                                            ELSIF (instMoveRelative.Error = TRUE) THEN
                                                statResetIncJog := TRUE;
                                                // Errorhandling
                                                statStatus                    := ERR_MC_MOVERELATIVE;
                                                statErrorAutoCleared          := TRUE;
                                                diagnostics                   := statDiagnostics;
                                                diagnostics.subfunctionStatus := instMoveRelative.ErrorId;
                                                // Set next state
                                                statFBState          := AXIS_STOP_ON_ERROR_SELECTION;
                                                statBasicMotionState := NO_SELECTION;
                                                statExeOfBasicMotion := CMD_ERROR;
                                                statIncJogSubState   := INC_JOG_IDLE;

                                            ELSIF (instMoveRelative.CommandAborted = TRUE) THEN
                                                statResetIncJog      := TRUE;
                                                statExeOfBasicMotion := CMD_ABORTED;
                                                statIncJogSubState   := INC_JOG_IDLE;

                                            ELSE
                                                // statJogDistance :=  axis.StatusPositioning.Distance;
                                                ; // Wait for next state
                                            END_IF;

                                        INC_JOG_STOP: // Executed if inputs are reset --> Stop jog operation OR if jogForward and jogBackward are set --> Error and stop axis
                                            instHalt(Axis := axis,
                                                     Execute := TRUE,
                                                     Deceleration := statDeceleration,
                                                     (*AbortAcceleration := FALSE,*)
                                                     Jerk := statJerk);

                                            // Evaluate MC_Command
                                            IF (instHalt.Done = TRUE) THEN
                                                // Set next state
                                                statExeOfBasicMotion := CMD_END_PROCESS;
                                                statIncJogSubState   := INC_JOG_IDLE;

                                            ELSIF (instHalt.Error = TRUE) THEN
                                                statResetIncJog := TRUE;
                                                // Errorhandling
                                                statStatus                    := ERR_MC_HALT;
                                                statErrorAutoCleared          := TRUE;
                                                diagnostics                   := statDiagnostics;
                                                diagnostics.subfunctionStatus := instHalt.ErrorId;
                                                // Set next state
                                                statFBState          := AXIS_STOP_ON_ERROR_SELECTION;
                                                statBasicMotionState := NO_SELECTION;
                                                statExeOfBasicMotion := CMD_ERROR;
                                                statIncJogSubState   := INC_JOG_IDLE;

                                            ELSIF (instHalt.CommandAborted = TRUE) THEN
                                                statResetIncJog := TRUE;
                                                // Set next state
                                                statIncJogSubState   := INC_JOG_IDLE;
                                                statExeOfBasicMotion := CMD_ABORTED;

                                            ELSE
                                                ; // Wait for stopping axis
                                            END_IF;

                                    ELSE
                                        // Errorhandling
                                        statStatus                    := ERR_UNDEFINED_INCREMENTAL_JOG_SUBSTATE;
                                        statErrorUserCleared          := TRUE;
                                        diagnostics                   := statDiagnostics;
                                        diagnostics.subfunctionStatus := 0;
                                        // Set errorstate
                                        statFBState := FB_ERROR;
                                    END_CASE;

                                CMD_DONE,
                                    CMD_ABORTED,
                                    CMD_ERROR,
                                    CMD_END_PROCESS:
                                    // Return to NO_SELECTION if command finished
                                    IF (statBasicCommand.2 = FALSE) AND (statBasicCommand.3 = FALSE)
                                        THEN
                                        // jogForward and jogbackward inputs are reset
                                        statExeOfBasicMotion := CMD_BUSY;
                                        statBasicMotionState := NO_SELECTION;
                                    ELSE
                                        ; // Wait for falling edge at inputs for jog
                                    END_IF;

                            ELSE
                                // Errorhandling
                                statStatus                    := ERR_UNDEFINED_INCREMENTAL_JOG_STATE;
                                statErrorUserCleared          := TRUE;
                                diagnostics.subfunctionStatus := 0;
                                diagnostics.basicMotionState  := statBasicMotionState;
                                // Set errorstate
                                statFBState := FB_ERROR;
                            END_CASE;
                    {END_REGION}

                    ELSE
                        // Errorhandling - Invalid jog state
                        statStatus                    := ERR_INVALID_JOG_MODE;
                        statErrorAutoCleared          := TRUE;
                        diagnostics                   := statDiagnostics;
                        diagnostics.subfunctionStatus := 0;
                        // Set next state
                        statFBState          := AXIS_STOP_ON_ERROR_SELECTION;
                        statBasicMotionState := NO_SELECTION;
                    END_CASE;
                {END_REGION}

                MOVE_VELOCITY_SELECTED:
                    // Additional features (applicative): Change setpoint on the fly (Velocity) 
                    {REGION "MOVEVELOCITY_SELECTED"}

                    // Firstcycle of command
                    IF (statFirstCycleBasicMotion = TRUE) THEN
                        // Reset MC_MOVEVELOCITY command
                        instMoveVelocity(Axis := axis,
                                         Execute := FALSE);

                        statVelocityChangeOnTheFly := configuration.moveVelocity.velocityChangeOnTheFly;
                        statVelocity               := configuration.moveVelocity.velocity;           // Store the last adjusted velocity value
                        statAcceleration           := configuration.moveVelocity.acceleration;       // Store the last adjusted acceleration value
                        statDeceleration           := configuration.moveVelocity.deceleration;       // Store the last adjusted deceleration value
                        statJerk                   := configuration.moveVelocity.jerk;               // Store the last adjusted jerk value 
                        statDirection              := configuration.moveVelocity.direction;          // Store the last adjusted axis direction 
                        statPositionControlled     := configuration.moveVelocity.positionControlled; // Store the last adjusted motion mode

                    ELSIF (statVelocityChangeOnTheFly = TRUE) AND
                        (configuration.moveVelocity.velocity <> statVelocity) // Velocity changed
                        AND
                        (instMoveVelocity.CommandAborted = FALSE)
                        THEN
                        // Reset MC_MOVEVELOCITY command
                        instMoveVelocity(Axis := axis,
                                         Execute := FALSE);

                        statVelocity := configuration.moveVelocity.velocity; // Store the last adjusted velocity value
                    END_IF;

                    // Call MC_Command
                    instMoveVelocity(Axis := axis,
                                     Execute := statBasicCommand.4 OR statFirstCycleBasicMotion, // Input: moveVelocity
                                     Velocity := statVelocity,
                                     Acceleration := statAcceleration,
                                     Deceleration := statDeceleration,
                                     Jerk := statJerk,
                                     Direction := statDirection,
                    (*PositionControlled :=  statPositionControlled,*)
                    (*Current := FALSE*) );

                    // Evaluate MC_Command
                    IF (instMoveVelocity.Busy = FALSE) AND
                        (instMoveVelocity.Error = FALSE) AND
                        (instMoveVelocity.CommandAborted = FALSE) AND
                        (instMoveVelocity.InVelocity = FALSE)
                        THEN
                        // Return to NO_SELECTION if command finished
                        statBasicMotionState := NO_SELECTION;

                    ELSIF (instMoveVelocity.Error = TRUE)
                        THEN
                        // Errorhandling
                        statStatus                    := ERR_MC_MOVEVELOCITY;
                        statErrorAutoCleared          := TRUE;
                        diagnostics                   := statDiagnostics;
                        diagnostics.subfunctionStatus := instMoveVelocity.ErrorId;
                        statVelocityChangeOnTheFly    := FALSE;
                        // Set next state
                        statFBState          := AXIS_STOP_ON_ERROR_SELECTION;
                        statBasicMotionState := NO_SELECTION;

                    ELSE
                        ; // Command selected
                    END_IF;

                    // Write MC_Command outputs to internal variable
                    statExeOfBasicMotion   := 16#0;
                    statExeOfBasicMotion.0 := instMoveVelocity.Busy;
                    statExeOfBasicMotion.2 := instMoveVelocity.CommandAborted;
                    statExeOfBasicMotion.3 := instMoveVelocity.Error;
                    statExeOfBasicMotion.4 := instMoveVelocity.InVelocity;
                {END_REGION}

                POS_RELATIVE_SELECTED:
                    // Additional features (applicative): Specified direction
                    {REGION "POS_RELATIVE_SELECTED"}
                    // Firstcycle of command
                    IF (statFirstCycleBasicMotion = TRUE) THEN
                        // Configurate the direction of rotation
                        // 
                        IF ((configuration.posRelative.direction = 0) AND (configuration.posRelative.distance >= 0.0)
                            ) // Sign of distance is evaluated
                            OR
                            (configuration.posRelative.direction = FORWARD_DIR) // Forward direction
                            THEN
                            statPosition := ABS(configuration.posRelative.distance);
                            // Reset MC_MOVERELATIVE command
                            instMoveRelative(Axis := axis,
                                             Execute := FALSE);

                            statApplicativeBasicMotionError := FALSE;

                        ELSIF ((configuration.posRelative.direction = 0) AND (configuration.posRelative.distance < 0.0)
                            ) // Sign of distance is evaluated
                            OR
                            (configuration.posRelative.direction = BACKWARD_DIR) // Backward direction
                            THEN
                            statPosition := -ABS(configuration.posRelative.distance);
                            // Reset MC_MOVERELATIVE command
                            instMoveRelative(Axis := axis,
                                             Execute := FALSE);

                            statApplicativeBasicMotionError := FALSE;

                        ELSE
                            // Errorhandling - Invalid direction
                            statStatus                      := ERR_INVALID_POS_RELATIVE_DIR;
                            statErrorAutoCleared            := TRUE;
                            diagnostics.subfunctionStatus   := 0;
                            diagnostics                     := statDiagnostics;
                            statApplicativeBasicMotionError := TRUE;
                            // Set next state
                            statFBState          := AXIS_STOP_ON_ERROR_SELECTION;
                            statBasicMotionState := NO_SELECTION;
                        END_IF;
                    END_IF;

                    IF (statApplicativeBasicMotionError = FALSE) THEN
                        // Call MC_Command
                        instMoveRelative(Axis := axis,
                                         Execute := statBasicCommand.5 OR statFirstCycleBasicMotion, // Input: posRelative
                                         Distance := statPosition,
                                         Velocity := configuration.posRelative.velocity,
                                         Acceleration := configuration.posRelative.acceleration,
                                         Deceleration := configuration.posRelative.deceleration,
                                         Jerk := configuration.posRelative.jerk);

                        // Evaluate MC_Command
                        IF (instMoveRelative.Busy = FALSE) AND
                            (instMoveRelative.Error = FALSE) AND
                            (instMoveRelative.Done = FALSE) AND
                            (instMoveRelative.CommandAborted = FALSE)
                            THEN
                            // Return to NO_SELECTION if command finished
                            statBasicMotionState := NO_SELECTION;

                        ELSIF (instMoveRelative.Error = TRUE) THEN
                            // Errorhandling
                            statStatus                    := ERR_MC_MOVERELATIVE;
                            statErrorAutoCleared          := TRUE;
                            diagnostics                   := statDiagnostics;
                            diagnostics.subfunctionStatus := instMoveRelative.ErrorId;
                            // Set next state
                            statFBState          := AXIS_STOP_ON_ERROR_SELECTION;
                            statBasicMotionState := NO_SELECTION;
                        ELSE
                            ; // Command selected
                        END_IF;

                        // Write MC_Command outputs to internal variable
                        statExeOfBasicMotion   := 16#0;
                        statExeOfBasicMotion.0 := instMoveRelative.Busy;
                        statExeOfBasicMotion.1 := instMoveRelative.Done;
                        statExeOfBasicMotion.2 := instMoveRelative.CommandAborted;
                        statExeOfBasicMotion.3 := instMoveRelative.Error;

                    ELSE
                        ; // Direction not valid
                    END_IF;
                {END_REGION}

                POS_ABSOLUTE_SELECTED:
                    // Additional features (applicative): Change setpoint on the fly (Velocity and Position)
                    {REGION "POS_ABSOLUTE_SELECTED"}
                    // Firstcycle of command
                    IF (statFirstCycleBasicMotion = TRUE) THEN
                        // Reset MC_MOVEABSOLUTE command
                        instMoveAbsolute(Axis := axis,
                                         Execute := FALSE);

                        statPosition     := configuration.posAbsolute.position;
                        statVelocity     := configuration.posAbsolute.velocity;     // Store the last adjusted velocity value
                        statAcceleration := configuration.posAbsolute.acceleration; // Store the last adjusted accerlation value
                        statDeceleration := configuration.posAbsolute.deceleration; // Store the last adjusted deceleration value
                        statJerk         := configuration.posAbsolute.jerk;         // Store the last adjusted jerk value
                        statDirection    := configuration.posAbsolute.direction;

                        statVelocityChangeOnTheFly := configuration.posAbsolute.velocityChangeOnTheFly;
                        statPositionChangeOnTheFly := configuration.posAbsolute.positionChangeOnTheFly;

                    ELSIF (((statVelocityChangeOnTheFly = TRUE) AND (configuration.posAbsolute.velocity <> statVelocity)) OR
                        ((statPositionChangeOnTheFly = TRUE) AND (configuration.posAbsolute.position <> statPosition))) AND
                        (instMoveAbsolute.CommandAborted = FALSE)
                        THEN
                        instMoveAbsolute(Axis := axis,
                                         Execute := FALSE);

                        IF (statVelocityChangeOnTheFly = TRUE) THEN // Apply the new velocity value
                            statVelocity := configuration.posAbsolute.velocity;
                        END_IF;

                        IF (statPositionChangeOnTheFly = TRUE) THEN // Apply the new position value
                            statPosition := configuration.posAbsolute.position;
                        END_IF;

                        // Reset MC_MOVEABSOLUTE command
                        instMoveAbsolute(Axis := axis,
                                         Execute := FALSE);
                    END_IF;

                    instMoveAbsolute(Axis := axis,
                                     Execute := statBasicCommand.6 OR statFirstCycleBasicMotion, // Input: posAbsolute
                                     Position := statPosition,
                                     Velocity := statVelocity,
                                     Acceleration := statAcceleration,
                                     Deceleration := statDeceleration,
                                     Jerk := statJerk,
                    (*Direction :=  statDirection*) );

                    // Evaluate MC_Command
                    IF (instMoveAbsolute.Busy = FALSE) AND
                        (instMoveAbsolute.Error = FALSE) AND
                        (instMoveAbsolute.Done = FALSE) AND
                        (instMoveAbsolute.CommandAborted = FALSE)
                        THEN
                        // Return to NO_SELECTION if command finished
                        statBasicMotionState := NO_SELECTION;

                    ELSIF (instMoveAbsolute.Error = TRUE) THEN
                        // Errorhandling
                        statStatus                    := ERR_MC_MOVEABSOLUTE;
                        statErrorAutoCleared          := TRUE;
                        diagnostics                   := statDiagnostics;
                        diagnostics.subfunctionStatus := instMoveAbsolute.ErrorId;
                        statVelocityChangeOnTheFly    := FALSE;
                        statPositionChangeOnTheFly    := FALSE;
                        // Set next state
                        statFBState          := AXIS_STOP_ON_ERROR_SELECTION;
                        statBasicMotionState := NO_SELECTION;

                    ELSE
                        ; // Command selected
                    END_IF;

                    // Write MC_Command outputs to internal variable
                    statExeOfBasicMotion   := 16#0;
                    statExeOfBasicMotion.0 := instMoveAbsolute.Busy;
                    statExeOfBasicMotion.1 := instMoveAbsolute.Done;
                    statExeOfBasicMotion.2 := instMoveAbsolute.CommandAborted;
                    statExeOfBasicMotion.3 := instMoveAbsolute.Error;
                {END_REGION}

                ACTIVE_HOMING_SELECTED:
                    // Additional fearure (applicative): homing on fixed stop
                    {REGION "ACTIVE_HOMING_SELECTED"}
                    // Firstcycle of command
                    IF (statFirstCycleBasicMotion = TRUE) THEN
                        statActiveHomingState  := configuration.homing.extendedMode;
                        statExeOfBasicMotion   := CMD_BUSY;
                        statPassiveHomingState := NO_HOMING_ACTIVE;
                    END_IF;

                    // Selection of extended homing mode  
                    CASE statActiveHomingState OF
                        STANDARD_HOMING:
                            // No additional features
                            {REGION "STANDARD_HOMING"}
                            // Firstcycle of command
                            IF (statFirstCycleBasicMotion = TRUE) THEN
                                // Reset MC_HOME command
                                instHome(Axis := axis,
                                         bCalibrationCam := homingSensor,
                                         Execute := FALSE);

                                // Reset TON command
                                instTimerTON(IN := FALSE,
                                             PT := configuration.homing.homeExecutionTimeLimit);
                            END_IF;

                            // Call MC_Command
                            instHome(Axis := axis,
                                     bCalibrationCam := homingSensor,
                                     Execute := statBasicCommand.10 OR statFirstCycleBasicMotion, // Input: homing
                                     Position := configuration.homing.position,
                            (*Mode :=  configuration.homing.mode*) );

                            //Call TON
                            instTimerTON(IN := TRUE,
                                         PT := configuration.homing.homeExecutionTimeLimit);

                            // Evaluate MC_Command
                            IF (instHome.Busy = FALSE) AND
                                (instHome.Done = FALSE) AND
                                (instHome.CommandAborted = FALSE) AND
                                (instHome.Error = FALSE)
                                THEN
                                // Return to NO_SELECTION if command finished
                                statActiveHomingState := STANDARD_HOMING;
                                statBasicMotionState  := NO_SELECTION;

                            ELSIF (instHome.Error = TRUE OR instTimerTON.Q) THEN
                                // Errorhandling
                                statStatus                    := ERR_MC_HOME;
                                statErrorAutoCleared          := TRUE;
                                diagnostics                   := statDiagnostics;
                                diagnostics.subfunctionStatus := instHome.ErrorId;
                                statFBState                   := AXIS_STOP_ON_ERROR_SELECTION;
                                statBasicMotionState          := NO_SELECTION;

                            ELSE
                                ; // Command selected

                            END_IF;

                            statExeOfBasicMotion   := 16#0;
                            statExeOfBasicMotion.0 := instHome.Busy;
                            statExeOfBasicMotion.1 := instHome.Done;
                            statExeOfBasicMotion.2 := instHome.CommandAborted;
                            statExeOfBasicMotion.3 := instHome.Error;
                        {END_REGION}
                        HOMING_ON_FIXED_STOP:
                            // This case is additional feature (MC_MOVEVELOCITY and MC_HOME internal used)
                            {REGION "REFERENCE_TO_FIXED_STOP"}
                            CASE statExeOfBasicMotion OF
                                CMD_BUSY:
                                    // Firstcycle of command
                                    IF (statFirstCycleBasicMotion = TRUE) THEN
                                        // Check if homing on fixed stop is allowed  
                                        (*IF ( axis.Modulo.Enable = TRUE) THEN*)
                                        IF (tempFalse = TRUE) THEN
                                            // Modulo enabled - Errorhandling
                                            statStatus                    := ERR_MODULO_NOT_ALLOWED;
                                            statErrorAutoCleared          := TRUE;
                                            diagnostics.subfunctionStatus := 0;
                                            diagnostics.basicMotionState  := statBasicMotionState;
                                            // Set next state
                                            statFBState           := AXIS_STOP_ON_ERROR_SELECTION;
                                            statBasicMotionState  := NO_SELECTION;
                                            statActiveHomingState := STANDARD_HOMING;
                                            statHomingSubState    := HOMING_IDLE;

                                        ELSIF (configuration.homing.extendedModeTorqueLimit = 0) // Torqueliming 0 in configuration 
                                            THEN
                                            // Errorhandling -  Torquevalue 0 configured
                                            statStatus                    := ERR_INVALID_TORQUE_LIMIT;
                                            statErrorAutoCleared          := TRUE;
                                            diagnostics.subfunctionStatus := 0;
                                            diagnostics.basicMotionState  := statBasicMotionState;
                                            // Set next state
                                            statFBState           := AXIS_STOP_ON_ERROR_SELECTION;
                                            statBasicMotionState  := NO_SELECTION;
                                            statActiveHomingState := STANDARD_HOMING;
                                            statHomingSubState    := HOMING_IDLE;

                                            (*ELSIF ( axis.Homing.ReferencingVelocity = 0)*)
                                        ELSIF (configuration.homing.offsetPositionVelocity = 0)
                                            THEN
                                            // Errorhandling -  Velocity 0 configured
                                            statStatus                    := ERR_INVALID_VELOCITY;
                                            statErrorAutoCleared          := TRUE;
                                            diagnostics.subfunctionStatus := 0;
                                            diagnostics.basicMotionState  := statBasicMotionState;
                                            // Set next state
                                            statFBState           := AXIS_STOP_ON_ERROR_SELECTION;
                                            statBasicMotionState  := NO_SELECTION;
                                            statActiveHomingState := STANDARD_HOMING;
                                            statHomingSubState    := HOMING_IDLE;

                                        ELSE
                                            // Store dynamic values
                                            (*statHomingPosition :=  configuration.homing.position;
	                             statVelocity :=  axis.Homing.ReferencingVelocity;
	                             statAcceleration :=  axis.DynamicDefaults.Acceleration;
	                             statDeceleration :=  axis.DynamicDefaults.Deceleration;
	                             statJerk :=  axis.DynamicDefaults.Jerk;
	                             statTorqueLimit :=  configuration.homing.extendedModeTorqueLimit;*)
                                            statHomingPosition := configuration.homing.position;
                                            statVelocity       := configuration.homing.offsetPositionVelocity;
                                            statAcceleration   := configuration.homing.offsetPositionAcceleration;
                                            statDeceleration   := configuration.homing.offsetPositonDeceleration;
                                            statJerk           := configuration.homing.offsetPositionJerk;
                                            statTorqueLimit    := configuration.homing.extendedModeTorqueLimit;

                                            // Detecting operating sensor
                                            (*
								FOR  tempIndex := 1 TO 4 DO
	                              IF  axis.StatusSensor[ tempIndex].Control = TRUE
	                              THEN
	                                EXIT;
	                              END_IF;
	                            END_FOR;
	                            *)
                                            (*IF ( axis.Sensor[ tempIndex].ActiveHoming.Direction = 0) // Positve direction configured
	                            THEN*)
                                            // Positive direction
                                            statDirection := FORWARD_DIR;
                                            (* ELSE
	                              // Negative direction
	                               statDirection :=  BACKWARD_DIR;
	                            END_IF;
	                            *)
                                            (*statTorqueLimitingState :=  FIXED_STOP_DETECTION_ACTIVE;*)
                                            // Reset MC_Commands
                                            instHome(Axis := axis,
                                                     bCalibrationCam := homingSensor,
                                                     Execute := FALSE);

                                            instMoveVelocity(Axis := axis,
                                                             Execute := FALSE);

                                            instMoveAbsolute(Axis := axis,
                                                             Execute := FALSE);

                                            // Reset TON
                                            instTimerTON(IN := FALSE,
                                                         PT := configuration.homing.homeExecutionTimeLimit);

                                            // Determine the encoder type
                                            (* tempIndex := 1;
	                             tempIndex := UDINT_TO_INT( axis.OperativeSensor);
	                            IF ( axis.Sensor[ tempIndex].Type =  INCREMENTAL_ENCODER) THEN
	                               statHomingMode :=  DIRECT_HOMING; // Direct homing (absolute)
	                            ELSE
	                               statHomingMode :=  ABSOLUTE_ENCODER_ADJUSTMENT;
	                            END_IF;
								*)
                                            // Use always direct homing
                                            // statHomingMode :=  DIRECT_HOMING; // Direct homing (absolute)
                                            // Set next state
                                            (*statHomingSubState :=  HOMING_FIXED_STOP_DETECTION;*)
                                            statHomingSubState := HOMING_PROCESS;
                                        END_IF;
                                    END_IF;

                                    // Call OF subStateMachine
                                    REPEAT
                                        CASE statHomingSubState OF
                                            HOMING_IDLE:
                                                tempStateChangeActive := FALSE;
                                                ; // Do nothing, inserted no exectution of homing if error occurred in first cycle

                                            HOMING_FIXED_STOP_DETECTION:
                                                tempStateChangeActive := FALSE;

                                                // Start axis to detect fixed stop
                                                instMoveVelocity(Axis := axis,
                                                                 Execute := TRUE,
                                                                 Velocity := statVelocity,
                                                                 Acceleration := statAcceleration,
                                                                 Deceleration := statDeceleration,
                                                                 Jerk := statJerk,
                                                (*PositionControlled := TRUE,*)
                                                (*Direction :=  statDirection*) );

                                                // Read Statusword only when not already read out
                                                IF (tempStatusWord = 16#0)
                                                    THEN
                                                    (*tempStatusWord :=  axis.StatusWord;*)
                                                    tempStatusWord := axis.NcToPlc.StateDWord;
                                                END_IF;

                                                // Evaluate MC_Command
                                                IF (tempStatusWord.30 = TRUE) THEN // inClamping = TRUE
                                                    // Fixed stop detected --> start homing process
                                                    statHomingSubState    := HOMING_PROCESS;
                                                    tempStateChangeActive := TRUE;

                                                ELSIF (instMoveVelocity.Error = TRUE) THEN
                                                    // Errorhandling
                                                    statStatus                    := ERR_MC_MOVEVELOCITY;
                                                    statErrorAutoCleared          := TRUE;
                                                    diagnostics                   := statDiagnostics;
                                                    diagnostics.subfunctionStatus := instMoveVelocity.ErrorId;
                                                    // Set next state
                                                    statFBState           := AXIS_STOP_ON_ERROR_SELECTION;
                                                    statBasicMotionState  := NO_SELECTION;
                                                    statActiveHomingState := STANDARD_HOMING;
                                                    statExeOfBasicMotion  := CMD_ERROR;
                                                    statHomingSubState    := HOMING_IDLE;

                                                ELSIF (instMoveVelocity.CommandAborted = TRUE) THEN
                                                    // Set next state
                                                    statExeOfBasicMotion := CMD_ABORTED;
                                                    statHomingSubState   := HOMING_IDLE;

                                                ELSE
                                                    ; // Wait for detecting fixed stop
                                                END_IF;

                                            HOMING_PROCESS:
                                                tempStateChangeActive := FALSE;
                                                // Execute MC_HOME
                                                instHome(Axis := axis,
                                                         bCalibrationCam := homingSensor,
                                                         Execute := TRUE,
                                                         Position := statHomingPosition,
                                                (*Mode :=  statHomingMode*) );

                                                //Call TON
                                                instTimerTON(IN := TRUE,
                                                             PT := configuration.homing.homeExecutionTimeLimit);

                                                // Evaluate MC_Command
                                                IF (instHome.Done = TRUE) THEN
                                                    // MC_HOME finished - Set next state
                                                    statHomingSubState    := HOMING_POSITION;
                                                    tempStateChangeActive := TRUE;
                                                    instTimerTON.IN       := FALSE;

                                                ELSIF (instHome.Error = TRUE OR instTimerTON.Q) THEN
                                                    // Errorhandling
                                                    statStatus                    := ERR_MC_HOME;
                                                    statErrorAutoCleared          := TRUE;
                                                    diagnostics                   := statDiagnostics;
                                                    diagnostics.subfunctionStatus := instHome.ErrorId;
                                                    // Set next state
                                                    statFBState          := AXIS_STOP_ON_ERROR_SELECTION;
                                                    statExeOfBasicMotion := CMD_ERROR;
                                                    statHomingSubState   := HOMING_IDLE;

                                                ELSIF (instHome.CommandAborted = TRUE) THEN
                                                    // Set next state
                                                    statExeOfBasicMotion := CMD_ABORTED;
                                                    statHomingSubState   := HOMING_IDLE;
                                                ELSE
                                                    ; // Wait for finish homing process
                                                END_IF;

                                            HOMING_POSITION:
                                                tempStateChangeActive := FALSE;

                                                statHomingPosition := configuration.homing.offsetPosition;
                                                statVelocity       := configuration.homing.offsetPositionVelocity;
                                                statAcceleration   := configuration.homing.offsetPositionAcceleration;
                                                statDeceleration   := configuration.homing.offsetPositonDeceleration;
                                                statJerk           := configuration.homing.offsetPositionJerk;

                                                // Execute moving to homeposition
                                                instMoveAbsolute(Axis := axis,
                                                                 Execute := TRUE,
                                                                 (*Position :=  statHomingPosition,*)
                                                                 Position := configuration.homing.offsetPosition,
                                                                 Velocity := ABS(statVelocity),
                                                                 Acceleration := statAcceleration,
                                                                 Deceleration := statDeceleration,
                                                                 Jerk := statJerk,
                                                (*Direction :=  SHORTEST_WAY_DIR*) );

                                                // Evaluate MC_Command
                                                IF (instMoveAbsolute.Done = TRUE) THEN
                                                    // Homeposition reached - Set next state
                                                    statExeOfBasicMotion := CMD_DONE;
                                                    statHomingSubState   := HOMING_IDLE;

                                                ELSIF (instMoveAbsolute.Error = TRUE) THEN
                                                    // Errorhandling
                                                    statStatus                    := ERR_MC_MOVEABSOLUTE;
                                                    statErrorAutoCleared          := TRUE;
                                                    diagnostics                   := statDiagnostics;
                                                    diagnostics.subfunctionStatus := instMoveAbsolute.ErrorId;
                                                    // Set next state
                                                    statFBState           := AXIS_STOP_ON_ERROR_SELECTION;
                                                    statBasicMotionState  := CMD_BUSY;
                                                    statActiveHomingState := STANDARD_HOMING;
                                                    statExeOfBasicMotion  := CMD_ERROR;
                                                    statHomingSubState    := HOMING_IDLE;

                                                ELSIF (instMoveAbsolute.CommandAborted = TRUE) THEN
                                                    // Set next state
                                                    statExeOfBasicMotion := CMD_ABORTED;
                                                    statHomingSubState   := HOMING_IDLE;

                                                ELSE
                                                    ; // Wait for reaching homeposition
                                                END_IF;

                                        ELSE
                                            // Errorhandling 
                                            statStatus                    := ERR_UNDEFINED_EXTENDED_HOMING_SUBSTATE;
                                            statErrorUserCleared          := TRUE;
                                            diagnostics                   := statDiagnostics;
                                            diagnostics.subfunctionStatus := 0;
                                            // Set errorstate
                                            statFBState           := FB_ERROR;
                                            tempStateChangeActive := FALSE;
                                        END_CASE;

                                    UNTIL (tempStateChangeActive = FALSE) // Repeat execution if a state is changing
                                    END_REPEAT;

                                CMD_DONE,
                                    CMD_ABORTED,
                                    CMD_ERROR:
                                    // Return to NO_SELECTION if command finished
                                    IF (statBasicCommand.10 = FALSE) // homing = FALSE
                                        THEN
                                        // Return to NO_HOMING_ACTIVE if command finished
                                        statBasicMotionState  := NO_SELECTION;
                                        statActiveHomingState := STANDARD_HOMING;
                                        statExeOfBasicMotion  := CMD_BUSY;
                                        statHomingSubState    := HOMING_IDLE;
                                    ELSE
                                        ; // Wait for falling edge at homing command
                                    END_IF;

                            ELSE
                                // Errorhandling
                                statStatus                    := ERR_UNDEFINED_EXTENDED_HOMING_STATE;
                                statErrorUserCleared          := TRUE;
                                diagnostics                   := statDiagnostics;
                                diagnostics.subfunctionStatus := 0;
                                // Set errorstate
                                statFBState := FB_ERROR;
                            END_CASE;
                    {END_REGION}

                    ELSE
                        // Errorhandling
                        statStatus                    := ERR_INVALID_HOMING_EXTENDED_MODE;
                        statErrorAutoCleared          := TRUE;
                        diagnostics                   := statDiagnostics;
                        diagnostics.subfunctionStatus := 0;
                        // Set next state
                        statFBState           := AXIS_STOP_ON_ERROR_SELECTION;
                        statBasicMotionState  := NO_SELECTION;
                        statActiveHomingState := STANDARD_HOMING;
                        statBasicMotionState  := NO_SELECTION;
                    END_CASE;
                {END_REGION}

                GEAR_IN_RELATIVE_SELECTED:
                    // Additional features (applicative): Change setpoint on the fly (gear ratio)
                    {REGION "GEAR_IN_RELATIVE_SELECTED"}
                    // Firstcycle of command
                    IF (statFirstCycleBasicMotion = TRUE) THEN
                        // Reset GEAR_IN command 
                        instGearIn(Master := master,
                                   Slave := axis,
                                   Execute := FALSE);

                        (*statRatioNumerator :=  configuration.gearInRelative.ratioNumerator;*)
                        statRatioNumerator      := configuration.gearInRelative.ratioDenominator;
                        statRatioDenominator    := configuration.gearInRelative.ratioDenominator;
                        statAcceleration        := configuration.gearInRelative.acceleration;
                        statDeceleration        := configuration.gearInRelative.deceleration;
                        statJerk                := configuration.gearInRelative.jerk;
                        statRatioChangeOnTheFly := configuration.gearInRelative.ratioChangeOnTheFly;

                    ELSIF ((statRatioChangeOnTheFly = TRUE) // Flying change of ratio numerator
                    (*AND (( configuration.gearInRelative.ratioNumerator <>  statRatioNumerator)*)
                        AND
                        ((configuration.gearInRelative.ratioDenominator <> statRatioNumerator) OR
                        (configuration.gearInRelative.ratioDenominator <> statRatioDenominator))) AND
                        (instGearIn.CommandAborted = FALSE)
                        THEN
                        instGearIn(Master := master,
                                   Slave := axis,
                                   Execute := FALSE);

                        statRatioNumerator   := configuration.gearInRelative.ratioDenominator; // Apply the new gear ratio numerator
                        statRatioDenominator := configuration.gearInRelative.ratioDenominator; // Apply the new gear ratio denominator
                    END_IF;

                    // Call MC_Command
                    instGearIn(Master := master,
                               Slave := axis,
                               Execute := statBasicCommand.7 OR statFirstCycleBasicMotion, // Input: gearInRelative
                               RatioNumerator := statRatioNumerator,
                               RatioDenominator := DINT_TO_UINT(statRatioDenominator),
                               Acceleration := statAcceleration,
                               Deceleration := statDeceleration,
                               Jerk := statJerk);

                    // Evaluate MC_Command
                    IF (instGearIn.Busy = FALSE) AND
                        (instGearIn.Error = FALSE) AND
                        (instGearIn.CommandAborted = FALSE) AND
                        (instGearIn.InGear = FALSE)
                        THEN
                        // Return to NO_SELECTION if command finished
                        statBasicMotionState := NO_SELECTION;

                    ELSIF (instGearIn.Error = TRUE) THEN
                        // Errorhandling
                        statStatus                    := ERR_MC_GEARIN;
                        statErrorAutoCleared          := TRUE;
                        diagnostics                   := statDiagnostics;
                        diagnostics.subfunctionStatus := instGearIn.ErrorId;
                        statRatioChangeOnTheFly       := FALSE;
                        // Set next state
                        statFBState          := AXIS_STOP_ON_ERROR_SELECTION;
                        statBasicMotionState := NO_SELECTION;

                    ELSE
                        ; // Command selected
                    END_IF;

                    // Read Statusword only when not already read out
                    // IF ( tempStatusWord = 16#0)
                    // THEN
                    //    tempStatusWord :=  axis.StatusWord;
                    // END_IF;

                    // Write MC_Command outputs to internal variable
                    statExeOfBasicMotion   := 16#0;
                    statExeOfBasicMotion.0 := instGearIn.Busy;
                    statExeOfBasicMotion.2 := instGearIn.CommandAborted;
                    statExeOfBasicMotion.3 := instGearIn.Error;
                    // statExeOfBasicMotion.6 :=  tempStatusWord.21 AND NOT  instGearIn.InGear; // write Synchronizing only when bit of instance of MC_GearIn.InGear = FALSE
                    statExeOfBasicMotion.7 := instGearIn.InGear;
                {END_REGION}

                GEAR_IN_ABSOLUTE_SELECTED:
                    // Additional features (applicative): Change setpoint on the fly (gear ratio)
                    {REGION "GEAR_IN_SELECTED"}
                    // Firstcycle of command
                    IF (statFirstCycleBasicMotion = TRUE) THEN
                        // Reset GEAR_IN_POS command 
                        instGearInPos(Master := master,
                                      Slave := axis,
                        (*Execute := FALSE*) );

                        statRatioNumerator       := configuration.gearInAbsolute.ratioNumerator;
                        statRatioDenominator     := configuration.gearInAbsolute.ratioDenominator;
                        statMasterSyncPosition   := configuration.gearInAbsolute.masterSyncPosition;
                        statSlaveSyncPosition    := configuration.gearInAbsolute.slaveSyncPosition;
                        statSyncProfileReference := configuration.gearInAbsolute.syncProfileReference;
                        statMasterStartDistance  := configuration.gearInAbsolute.masterStartDistance;
                        statVelocity             := configuration.gearInAbsolute.velocity;
                        statAcceleration         := configuration.gearInAbsolute.acceleration;
                        statDeceleration         := configuration.gearInAbsolute.deceleration;
                        statJerk                 := configuration.gearInAbsolute.jerk;
                        statSyncDirection        := configuration.gearInAbsolute.syncDirection;
                        statRatioChangeOnTheFly  := configuration.gearInAbsolute.ratioChangeOnTheFly;

                    ELSIF (((statRatioChangeOnTheFly = TRUE) AND (configuration.gearInAbsolute.ratioNumerator <> statRatioNumerator)) OR
                        ((statRatioChangeOnTheFly = TRUE) AND (configuration.gearInAbsolute.ratioDenominator <> statRatioDenominator))) AND
                        (instGearInPos.CommandAborted = FALSE)
                        THEN
                        instGearInPos(Master := master,
                                      Slave := axis,
                        (*Execute := FALSE*) );

                        statRatioNumerator   := configuration.gearInAbsolute.ratioNumerator;   // Apply the new gear ratio numerator
                        statRatioDenominator := configuration.gearInAbsolute.ratioDenominator; // Apply the new gear ratio denominator
                    END_IF;

                    // Call MC_Command
                    instGearInPos(Master := master,
                                  Slave := axis,
                                  Enable := statBasicCommand.8 OR statFirstCycleBasicMotion, // Input: gearInAbsolute
                                  GearRatio := statRatioNumerator,
                                  (*RatioDenominator :=  statRatioDenominator,*)
                                  (*MasterSyncPosition :=  statMasterSyncPosition,*)
                                  (*SlaveSyncPosition :=  statSlaveSyncPosition,*)
                                  (*SyncProfileReference :=  statSyncProfileReference,*)
                                  (*MasterStartDistance :=  statMasterStartDistance,*)
                                  (*Velocity :=  statVelocity,*)
                                  (*Acceleration :=  statAcceleration,*)
                                  (*Deceleration :=  statDeceleration,*)
                                  Jerk := statJerk,
                    (*SyncDirection :=  statSyncDirection*) );

                    // Evaluate MC_Command
                    IF (instGearInPos.Busy = FALSE) AND
                        (instGearInPos.Error = FALSE) AND
                        (instGearInPos.CommandAborted = FALSE) AND
                    (*( instGearInPos.StartSync = FALSE) AND*)
                        (instGearInPos.InGear = FALSE)
                        THEN
                        // Return to NO_SELECTION if command finished
                        statBasicMotionState := NO_SELECTION;

                    ELSIF (instGearInPos.Error = TRUE) THEN
                        // Errorhandling
                        statStatus                    := ERR_MC_GEARINPOS;
                        statErrorAutoCleared          := TRUE;
                        diagnostics                   := statDiagnostics;
                        diagnostics.subfunctionStatus := instGearInPos.ErrorId;
                        statRatioChangeOnTheFly       := FALSE;
                        // Set next state
                        statFBState          := AXIS_STOP_ON_ERROR_SELECTION;
                        statBasicMotionState := NO_SELECTION;

                    ELSE
                        ; // Command selected
                    END_IF;

                    // Write MC_Command outputs to internal variable
                    statExeOfBasicMotion   := 16#0;
                    statExeOfBasicMotion.0 := instGearInPos.Busy;
                    statExeOfBasicMotion.2 := instGearInPos.CommandAborted;
                    statExeOfBasicMotion.3 := instGearInPos.Error;
                    (*statExeOfBasicMotion.6 :=  instGearInPos.StartSync;*)
                    (*statExeOfBasicMotion.6 :=  instGearInPos.StartSync;*)
                    statExeOfBasicMotion.7 := instGearInPos.InGear;
                {END_REGION}

                CAM_IN_SELECTED:
                    // Additional feature (applicative): Check DB of Cam 
                    {REGION "CAM_IN_SELECTED"}
                    // Firstcycle of command
                    IF (statFirstCycleBasicMotion = TRUE) THEN
                        (*IF TypeOfDB( cam) = TO_Cam*)
                        IF tempFalse = FALSE
                            THEN
                            (*statCam :=  cam;*)
                            // Reset CAM_IN command 
                            instCamIn(Master := master,
                                      Slave := axis,
                                      (*Cam :=  statCam,*)
                                      Execute := FALSE);

                            statApplicativeBasicMotionError := FALSE;
                            statApplicationMode             := configuration.camIn.applicationMode;
                        ELSE
                            // Errorhandling - Invalid cam
                            statStatus                      := ERR_INVALID_CAM;
                            statErrorAutoCleared            := TRUE;
                            diagnostics.subfunctionStatus   := 0;
                            diagnostics                     := statDiagnostics;
                            statApplicativeBasicMotionError := TRUE;
                            // Set next state
                            statFBState          := AXIS_STOP_ON_ERROR_SELECTION;
                            statBasicMotionState := NO_SELECTION;
                        END_IF;
                    END_IF;

                    IF (statApplicativeBasicMotionError = FALSE) THEN

                        // Write MC Parameters
                        instCamIn.CamTableID                 := configuration.camIn.tableID;
                        instCamIn.StartMode                  := configuration.camIn.startMode;
                        instCamIn.MasterOffset               := configuration.camIn.masterOffset;
                        instCamIn.SlaveOffset                := configuration.camIn.slaveOffset;
                        instCamIn.MasterScaling              := configuration.camIn.masterScaling;
                        instCamIn.SlaveScaling               := configuration.camIn.slaveScaling;
						instCamIn.StartMode     			 := configuration.camIn.startMode;
                        instCamIn.Options.ActivationMode     := configuration.camIn.ActivationMode;
                        instCamIn.Options.ActivationPosition := configuration.camIn.ActivationPosition;

                        // Call MC_Command
                        instCamIn(Master := master,
                                  Slave := axis,
                                  Execute := statBasicCommand.9 OR statFirstCycleBasicMotion);

                        // Evaluate MC_Command
                        IF ((instCamIn.Busy = FALSE) AND
                            (instCamIn.Error = FALSE) AND
                            (instCamIn.CommandAborted = FALSE) AND
                            (instCamIn.InSync = FALSE) AND
                        (*( instCamIn.StartSync = FALSE) AND*)
                            (statBasicCommand.9 = FALSE)
                            ) AND // V1.0.2 Wait for one cycle EndOfProfile (--> Done) before function is finished at applicationMode ONCE
                            ((statApplicationMode <> APPLICATION_MODE_ONCE) OR
                            ((statApplicationMode = APPLICATION_MODE_ONCE) (*AND ( instCamIn.EndOfProfile = FALSE)*) ))
                            THEN
                            // Return to NO_SELECTION if command finished
                            statBasicMotionState := NO_SELECTION;

                        ELSIF (instCamIn.Error = TRUE) THEN
                            // Errorhandling
                            statStatus                    := ERR_MC_CAMIN;
                            statErrorAutoCleared          := TRUE;
                            diagnostics.subfunctionStatus := instCamIn.ErrorId;
                            diagnostics.basicMotionState  := statBasicMotionState;
                            statFBState                   := AXIS_STOP_ON_ERROR_SELECTION;
                            statBasicMotionState          := NO_SELECTION;

                        ELSE
                            ; // Command selected
                        END_IF;

                        // Write MC_Command outputs to internal variable
                        statExeOfBasicMotion   := 16#0;
                        statExeOfBasicMotion.0 := instCamIn.Busy;
                        IF (statApplicationMode = APPLICATION_MODE_ONCE)
                            THEN
                            ; (*statExeOfBasicMotion.1 :=  instCamIn.EndOfProfile;*)
                        END_IF;

                        statExeOfBasicMotion.2 := instCamIn.CommandAborted;
                        statExeOfBasicMotion.3 := instCamIn.Error;
                        statExeOfBasicMotion.6 := NOT instCamIn.Active;
                        statExeOfBasicMotion.7 := instCamIn.InSync;

                    ELSE
                        ; // InValid cam
                    END_IF;
            {END_REGION}

            ELSE
                // Errorhandling
                statStatus                    := ERR_UNDEFINED_BASIC_MOTION_STATE;
                statErrorUserCleared          := TRUE;
                diagnostics                   := statDiagnostics;
                diagnostics.subfunctionStatus := 0;
                // Set errorstate
                statFBState := FB_ERROR;
            END_CASE;

        RESET_GEARING:
            // Abort waiting absolute gearing / camIn job if new basic motion job is selected (configuration.generalSettings.abortWaitingSyncCmd = TRUE)
            instGearIn(Master := master,
                       Slave := axis,
                       Execute := TRUE,
                       RatioNumerator := 1,
                       RatioDenominator := 1); // Lowest possible gear ratio

            IF (instGearIn.InGear = TRUE) OR (instGearIn.CommandAborted = TRUE)
                THEN                                            // Relative gearing command has aborted waiting absolute gearing job
                statMainSelectionState    := CALL_BASIC_MOTION; // Execute new basic motion command
                tempStateChangeActive     := TRUE;
                statFirstCycleBasicMotion := TRUE;

            ELSIF (instGearIn.Error = TRUE)
                THEN
                statStatus                    := ERR_MC_GEARIN;
                diagnostics.subfunctionStatus := instGearIn.ErrorId;
                // Errorhandling
                statErrorAutoCleared := TRUE;
                diagnostics          := statDiagnostics;
                // Set next state
                statFBState            := AXIS_STOP_ON_ERROR_SELECTION;
                statMainSelectionState := CALL_BASIC_MOTION;
                statBasicMotionState   := NO_SELECTION;

            ELSE
                ; // Command running
            END_IF;

            // Write MC_Command outputs to internal variable
            statExeOfBasicMotion   := 16#0;
            statExeOfBasicMotion.0 := instGearIn.Busy;
    ELSE
        // Errorhandling
        statStatus                    := ERR_UNDEFINED_MAIN_SELECTION_STATE;
        statErrorUserCleared          := TRUE;
        diagnostics                   := statDiagnostics;
        diagnostics.subfunctionStatus := 0;
        // Set errorstate
        statFBState := FB_ERROR;
    END_CASE;

UNTIL (tempStateChangeActive = FALSE)
END_REPEAT;

{END_REGION}

//----------------------------------------------------------------------------------------------
// Execution of homing functionality 
//----------------------------------------------------------------------------------------------
{REGION "EXECUTION_OF_PASSIVE_HOMING"}
// Statemachine for homing functionality
CASE statPassiveHomingState OF
    // Selection of extended homing mode  
    NO_HOMING_ACTIVE:
        ; // Do nothing

    STANDARD_HOMING:
        // No additional features
        {REGION "STANDARD_HOMING"}
        // Firstcycle of command
        IF (statFirstCycleHoming = TRUE) THEN
            // Reset MC_HOME command
            instHome(Axis := axis,
                     bCalibrationCam := homingSensor,
                     Execute := FALSE);

            IF (statBasicMotionState = ACTIVE_HOMING_SELECTED) THEN
                statBasicMotionState := NO_SELECTION;
            END_IF;
        END_IF;

        // Call MC_Command
        instHome(Axis := axis,
                 bCalibrationCam := homingSensor,
                 Execute := statExtendedCommand.2, // Input: homing
                 Position := configuration.homing.position,
        (*Mode :=  configuration.homing.mode*) );

        // Evaluate MC_Command
        IF (instHome.Busy = FALSE) AND
            (instHome.Done = FALSE) AND
            (instHome.CommandAborted = FALSE) AND
            (instHome.Error = FALSE)
            THEN
            // Return to NO_SELECTION if command finished
            statPassiveHomingState := NO_HOMING_ACTIVE;

        ELSIF (instHome.Error = TRUE) THEN
            // Errorhandling
            statStatus                    := ERR_MC_HOME;
            statErrorAutoCleared          := TRUE;
            diagnostics                   := statDiagnostics;
            diagnostics.subfunctionStatus := instHome.ErrorId;
            statPassiveHomingState        := NO_HOMING_ACTIVE;
            // Set next state
            statFBState := AXIS_STOP_ON_ERROR_SELECTION;
        ELSE
            ; // Command selected

        END_IF;

        statExeOfHoming   := 16#0;
        statExeOfHoming.0 := instHome.Busy;
        statExeOfHoming.1 := instHome.Done;
        statExeOfHoming.2 := instHome.CommandAborted;
        statExeOfHoming.3 := instHome.Error;
{END_REGION}

ELSE
    // Errorhandling
    statStatus                              := ERR_INVALID_HOMING_EXTENDED_MODE;
    statErrorAutoCleared                    := TRUE;
    diagnostics                             := statDiagnostics;
    diagnostics.subfunctionStatus           := 0;
    statDiagnostics.basicMotionState        := statBasicMotionState;
    statDiagnostics.superimposedMotionState := statSupImpMotionState;
    // Set next state
    statFBState            := AXIS_STOP_ON_ERROR_SELECTION;
    statBasicMotionState   := NO_SELECTION;
    statPassiveHomingState := NO_HOMING_ACTIVE;
END_CASE;

{END_REGION}

//----------------------------------------------------------------------------------------------
// Execution of functionalities of superimposed coordinate system
//----------------------------------------------------------------------------------------------
{REGION "EXECUTION_OF_SUPERIMPOSED_COMMANDS"}
// Statemachine for superimposed motion commands
// Write diagnostics
statDiagnostics.basicMotionState        := statBasicMotionState;
statDiagnostics.superimposedMotionState := statSupImpMotionState;

CASE statSupImpMotionState OF
    NO_SELECTION:
        ; // Do nothing

    POS_SUPERIMPOSED_SELECTED:
        // Additional features (applicative) : Specified direction
        {REGION "POS_SUPERIMPOSED_SELECTED;"}
        // Firstcycle of command
        IF (statFirstCycleSupImpMotion = TRUE) THEN
            // Configurate the direction of rotation
            IF ((configuration.posSuperimposed.direction = 0) AND (configuration.posSuperimposed.distance >= 0.0)) // Sign of distance is evaluated
                OR
                (configuration.posSuperimposed.direction = FORWARD_DIR) // Positive direction
                THEN
                statSupImpMotionPosition := ABS(configuration.posSuperimposed.distance);
                // Reset MC_MOVESUPERIMPOSED command
                instMoveSuperimposed(Axis := axis,
                                     Execute := FALSE);

                statApplicativeSupImpMotionError := FALSE;
            ELSIF ((configuration.posSuperimposed.direction = 0) AND (configuration.posSuperimposed.distance < 0.0)) // Sign of distance is evaluated
                OR
                (configuration.posSuperimposed.direction = BACKWARD_DIR) // Negative direction 
                THEN
                statSupImpMotionPosition := -ABS(configuration.posSuperimposed.distance);
                // Reset MC_MOVESUPERIMPOSED command
                instMoveSuperimposed(Axis := axis,
                                     Execute := FALSE);

                statApplicativeSupImpMotionError := FALSE;

            ELSE
                // Errorhandling - Invalid direction
                statStatus                       := ERR_INVALID_POS_SUPERIMPOSED_DIR;
                statErrorAutoCleared             := TRUE;
                diagnostics                      := statDiagnostics;
                diagnostics.subfunctionStatus    := 0;
                statApplicativeSupImpMotionError := TRUE;
                // Set next state
                statFBState           := AXIS_STOP_ON_ERROR_SELECTION;
                statSupImpMotionState := NO_SELECTION;
            END_IF;
        END_IF;

        IF (statApplicativeSupImpMotionError = FALSE) THEN
            // Call MC_Command
            instMoveSuperimposed(Axis := axis,
                                 Execute := statSupImpCommand.0, // Input: posSuperimposed
                                 Distance := statSupImpMotionPosition,
                                 VelocityDiff := configuration.posSuperimposed.velocityDiff,
                                 Acceleration := configuration.posSuperimposed.acceleration,
                                 Deceleration := configuration.posSuperimposed.deceleration,
                                 Jerk := configuration.posSuperimposed.jerk);

            // Evaluate MC_Command
            IF (instMoveSuperimposed.Busy = FALSE) AND
                (instMoveSuperimposed.Error = FALSE) AND
                (instMoveSuperimposed.Done = FALSE) AND
                (instMoveSuperimposed.CommandAborted = FALSE)
                THEN
                // Return to NO_SELECTION if command finished
                statSupImpMotionState := NO_SELECTION;

            ELSIF (instMoveSuperimposed.Error = TRUE) THEN
                // Errorhandling
                statStatus                    := ERR_MC_MOVESUPERIMPOSED;
                statErrorAutoCleared          := TRUE;
                diagnostics                   := statDiagnostics;
                diagnostics.subfunctionStatus := instMoveSuperimposed.ErrorId;
                // Set next state
                statFBState           := AXIS_STOP_ON_ERROR_SELECTION;
                statSupImpMotionState := NO_SELECTION;

            ELSE
                ; // command selected
            END_IF;

            statExeOfSupImpMotionState   := 16#0;
            statExeOfSupImpMotionState.0 := instMoveSuperimposed.Busy;
            statExeOfSupImpMotionState.1 := instMoveSuperimposed.Done;
            statExeOfSupImpMotionState.2 := instMoveSuperimposed.CommandAborted;
            statExeOfSupImpMotionState.3 := instMoveSuperimposed.Error;
        END_IF;
    {END_REGION}

    PHASING_SELECTED:
        // Additional features (applicative) : Change setpoint on the fly (phaseShift)
        {REGION "PHASING_SELECTED"}
        // Firstcycle of command
        IF (statFirstCycleSupImpMotion = TRUE) THEN
            // Reset MC_PHASING_ABSOLUTE command
            instPhasingAbsolute(Master := master,
                                Slave := axis,
                                Execute := FALSE);

            // Reset MC_PHASING_RELATIVE command
            instPhasingRelative(Master := master,
                                Slave := axis,
                                Execute := FALSE);

            statPhaseShift               := configuration.phasing.phaseShift;
            statVelocity                 := configuration.phasing.velocity;
            statAcceleration             := configuration.phasing.acceleration;
            statDeceleration             := configuration.phasing.deceleration;
            statJerk                     := configuration.phasing.jerk;
            statPhaseAbsolute            := configuration.phasing.phaseAbsolute;
            statChangePhaseShiftOnTheFly := configuration.phasing.phaseShiftChangeOnTheFly;

        ELSIF ((statChangePhaseShiftOnTheFly = TRUE) AND
            (configuration.phasing.phaseShift <> statPhaseShift)) AND
            (statPhaseAbsolute = TRUE) AND
            (instPhasingAbsolute.CommandAborted = FALSE)
            THEN
            // Reset MC_PHASING_ABSOLUTE command - Phaseshift on the fly is only possible at phasing absolut
            instPhasingAbsolute(Master := master,
                                Slave := axis,
                                Execute := FALSE);

            statPhaseShift := configuration.phasing.phaseShift;
        END_IF;

        // Select phasing absolut or relative 
        IF (statPhaseAbsolute = TRUE) THEN
            // Absolute phasing
            // Call MC_Command
            instPhasingAbsolute(Master := master,
                                Slave := axis,
                                Execute := statSupImpCommand.1, // Input: phasing
                                PhaseShift := statPhaseShift,
                                Velocity := statVelocity,
                                Acceleration := statAcceleration,
                                Deceleration := statDeceleration,
                                Jerk := statJerk);

            // Evaluate MC_Command
            IF (instPhasingAbsolute.Busy = FALSE) AND
                (instPhasingAbsolute.Error = FALSE) AND
                (instPhasingAbsolute.Done = FALSE) AND
                (instPhasingAbsolute.CommandAborted = FALSE)
                THEN
                // Return to NO_SELECTION if command finished
                statSupImpMotionState := NO_SELECTION;

            ELSIF (instPhasingAbsolute.Error = TRUE) THEN
                // Errorhandling
                statStatus                    := ERR_MC_PHASINGABSOLUTE;
                statErrorAutoCleared          := TRUE;
                diagnostics                   := statDiagnostics;
                diagnostics.subfunctionStatus := instPhasingAbsolute.ErrorId;
                statChangePhaseShiftOnTheFly  := FALSE;
                // Set next state
                statFBState           := AXIS_STOP_ON_ERROR_SELECTION;
                statSupImpMotionState := NO_SELECTION;

            ELSE
                ; // Command busy
            END_IF;

            statExeOfSupImpMotionState   := 16#0;
            statExeOfSupImpMotionState.0 := instPhasingAbsolute.Busy;
            statExeOfSupImpMotionState.1 := instPhasingAbsolute.Done;
            statExeOfSupImpMotionState.2 := instPhasingAbsolute.CommandAborted;
            statExeOfSupImpMotionState.3 := instPhasingAbsolute.Error;

        ELSE
            // Relative phasing  
            // Call MC_Command
            instPhasingRelative(Master := master,
                                Slave := axis,
                                Execute := statSupImpCommand.1, // Input: phasing
                                PhaseShift := statPhaseShift,
                                Velocity := statVelocity,
                                Acceleration := statAcceleration,
                                Deceleration := statDeceleration,
                                Jerk := statJerk);

            // Evaluate MC_Command
            IF (instPhasingRelative.Busy = FALSE) AND
                (instPhasingRelative.Error = FALSE) AND
                (instPhasingRelative.Done = FALSE) AND
                (instPhasingRelative.CommandAborted = FALSE)
                THEN
                // Return to NO_SELECTION if command finished
                statSupImpMotionState := NO_SELECTION;

            ELSIF (instPhasingRelative.Error = TRUE) THEN
                // Errorhandling
                statStatus                    := ERR_MC_PHASINGRELATIVE;
                statErrorAutoCleared          := TRUE;
                diagnostics                   := statDiagnostics;
                diagnostics.subfunctionStatus := instPhasingRelative.ErrorId;
                statChangePhaseShiftOnTheFly  := FALSE;
                // Set next state
                statFBState           := AXIS_STOP_ON_ERROR_SELECTION;
                statSupImpMotionState := NO_SELECTION;
            ELSE
                ; // Command selected
            END_IF;

            statExeOfSupImpMotionState   := 16#0;
            statExeOfSupImpMotionState.0 := instPhasingRelative.Busy;
            statExeOfSupImpMotionState.1 := instPhasingRelative.Done;
            statExeOfSupImpMotionState.2 := instPhasingRelative.CommandAborted;
            statExeOfSupImpMotionState.3 := instPhasingRelative.Error;
        END_IF;
{END_REGION}

ELSE
    // Errorhandling
    statStatus                    := ERR_UNDEFINED_SUPERIMPOSED_MOTION_STATE;
    statErrorUserCleared          := TRUE;
    diagnostics                   := statDiagnostics;
    diagnostics.subfunctionStatus := 0;
    // Set errorstate
    statFBState := FB_ERROR;
END_CASE;

{END_REGION}

//----------------------------------------------------------------------------------------------
// Execution of torquelimiting functionality
//----------------------------------------------------------------------------------------------
{REGION "EXECUTION_OF_TORQUELIMTING"}
// Statemachine for torquelimiting 
REPEAT
    tempStateChangeActive := FALSE;
    CASE statTorqueLimitingState OF
        NO_TORQUE_LIMITING_ACTIVE:
            ; // Torquelimiting disable
        //  instTorqueLimiting(Axis :=  axis, V01.00.03 Dont Call MC_TORQUELIMITING if disabled
        //                     Enable := FALSE);

        TORQUE_LIMITING_DISABLE:
            // Torquelimiting disable
            instTorqueLimiting(Axis := axis,
                               Enable := FALSE);

            // Check state of torque limting
            IF (instTorqueLimiting.Busy = FALSE)
                THEN
                // set next state
                statTorqueLimitingState := NO_TORQUE_LIMITING_ACTIVE;
            ELSE
                ; // Waiting for MC_Torquelimiting is not busy
            END_IF;

        TORQUE_LIMTING_SELECTED:
            // No extended homing function active
            instTorqueLimiting(Axis := axis,
                               Enable := statExtendedCommand.1,
                               TLimit := configuration.torqueLimiting.TorqueLimit,
                               Mode := configuration.torqueLimiting.mode);

            IF (instTorqueLimiting.Busy = FALSE) THEN
                // Reset state
                statTorqueLimitingState := NO_TORQUE_LIMITING_ACTIVE;
            END_IF;

        (*
	        V1.00.03 Not required anymore
	       AUTOMATIC_MODE_CHANGE:
	        // In this state the torquelimiting function is operating with Mode 1 (Fixed stop detection) until inClamping = FALSE
	         instTorqueLimiting(Axis :=  axis,
	                            Enable := TRUE,
	                            Limit :=  configuration.homing.extendedModeTorqueLimit); // V01.00.03 Always use configured value
	        
	        IF ( configuration.torqueLimiting.mode =  MODE_FIXED_STOP_DETECTION)
	          OR ( instTorqueLimiting.InClamping = FALSE)
	        THEN
	          // Change state
	           statTorqueLimitingState :=  TORQUE_LIMTING_SELECTED;
	           tempStateChangeActive := TRUE;
	        ELSE
	          ; // Wait for InClamping = FALSE
	        END_IF;
	        *)

        FIXED_STOP_DETECTION_ACTIVE:
            // Extended homing function active
            instTorqueLimiting(Axis := axis,
                               Enable := TRUE,
                               TLimit := configuration.homing.extendedModeTorqueLimit, // V01.00.03 Always use configured value
                               Mode := MODE_FIXED_STOP_DETECTION);

            IF ((statHomingSubState = HOMING_IDLE) AND (statBasicMotionState = ACTIVE_HOMING_SELECTED))
                THEN
                // Fixed stop process has finished - Axis is still in clamping
                statTorqueLimitingState := FIXED_STOP_DETECTION_FINISHED;
                tempStateChangeActive   := TRUE;

            ELSIF (statBasicMotionState <> ACTIVE_HOMING_SELECTED)
                THEN
                // Error occurred - change state depending on inClamping
                IF (instTorqueLimiting.InClamping = TRUE)
                    THEN
                    // Axis is in clamping
                    statTorqueLimitingState := FIXED_STOP_DETECTION_ERROR_IN_CLAMPING;
                    tempStateChangeActive   := TRUE;
                ELSE
                    // Axis is in not clamping
                    statTorqueLimitingState := FIXED_STOP_DETECTION_ERROR_NOT_IN_CLAMPING;
                    tempStateChangeActive   := TRUE;
                END_IF;

            ELSE
                ; // Fixed stop detection is running
            END_IF;

        FIXED_STOP_DETECTION_FINISHED:
            // Homing on fixed stop process has finished
            instTorqueLimiting(Axis := axis,
                               Enable := TRUE,
                               TLimit := configuration.homing.extendedModeTorqueLimit, // V01.00.03 Always use configured value
                               Mode := MODE_FIXED_STOP_DETECTION);

            IF (instTorqueLimiting.InClamping = FALSE)
                THEN
                // InClamping = FALSE
                IF (statExtendedCommand.1 = TRUE) // Torquelimiting
                    THEN
                    statTorqueLimitingState := TORQUE_LIMTING_SELECTED;
                ELSE
                    statTorqueLimitingState := TORQUE_LIMITING_DISABLE;
                END_IF;

                tempStateChangeActive := TRUE;
            ELSE
                // InClamping = TRUE
                IF (statExtendedCommand.1 = TRUE) // Torquelimiting
                    AND
                    (configuration.torqueLimiting.mode = MODE_FIXED_STOP_DETECTION)
                    THEN
                    // Change State
                    statTorqueLimitingState := TORQUE_LIMTING_SELECTED;
                    tempStateChangeActive   := TRUE;
                ELSE
                    ; // Wait for inClamping = FALSE
                END_IF;
            END_IF;

        FIXED_STOP_DETECTION_ERROR_IN_CLAMPING:
            // Errorstate, torquelimiting is still active and axis not in clamping
            instTorqueLimiting(Axis := axis,
                               Enable := TRUE,
                               TLimit := configuration.homing.extendedModeTorqueLimit, // V01.00.03 Always use configured value
                               Mode := MODE_FIXED_STOP_DETECTION);

            IF (instTorqueLimiting.InClamping = FALSE)
                THEN
                // InClamping = FALSE -> reset torque limiting state
                statTorqueLimitingState := TORQUE_LIMITING_DISABLE;
                // Torquelimiting disable
                tempStateChangeActive := TRUE;
            END_IF;

        FIXED_STOP_DETECTION_ERROR_NOT_IN_CLAMPING:
            // Errorstate, torquelimiting is still active and axis in clamping
            instTorqueLimiting(Axis := axis,
                               Enable := TRUE,
                               TLimit := configuration.homing.extendedModeTorqueLimit, // V01.00.03 Always use configured value
                               Mode := MODE_FIXED_STOP_DETECTION);

            IF (instTorqueLimiting.InClamping = TRUE)
                THEN
                // InClamping = TRUE -> change state
                statTorqueLimitingState := FIXED_STOP_DETECTION_ERROR_IN_CLAMPING;
                tempStateChangeActive   := TRUE;

            ELSIF (statBasicMotionState <> NO_SELECTION) OR (statSupImpMotionState <> NO_SELECTION) OR (statPassiveHomingState <> NO_HOMING_ACTIVE)
                THEN
                // New valid command is set -> reset error state
                statTorqueLimitingState := TORQUE_LIMITING_DISABLE;
                tempStateChangeActive   := TRUE;

            ELSE
                ; // Waiting for new command or axis is getting in clamping
            END_IF;
    ELSE
        // Errorhandling
        statStatus                          := ERR_UNDEFINED_TORQUE_LIMITING_STATE;
        statErrorUserCleared                := TRUE;
        diagnostics.basicMotionState        := statBasicMotionState;
        diagnostics.superimposedMotionState := statSupImpMotionState;
        diagnostics.subfunctionStatus       := 0;
        // Set errorstate
        statFBState := FB_ERROR;
    END_CASE;
UNTIL (tempStateChangeActive = FALSE)
END_REPEAT;

// Evaluate MC_Command
IF (instTorqueLimiting.Error = TRUE) AND ((statTorqueLimitingErrorOld = FALSE) OR (statStatus = STATUS_SUBSEQUENT_CALL)) THEN
    // Errorhandling
    statStatus                          := ERR_MC_TORQUELIMITING;
    statErrorAutoCleared                := TRUE;
    diagnostics.basicMotionState        := statBasicMotionState;
    diagnostics.superimposedMotionState := statSupImpMotionState;
    diagnostics.subfunctionStatus       := instTorqueLimiting.ErrorId;
    statFBState                         := AXIS_STOP_ON_ERROR_SELECTION;

ELSIF (instTorqueLimiting.Error = FALSE) AND ((statTorqueLimitingErrorOld = TRUE) AND (statStatus = ERR_MC_TORQUELIMITING)) THEN
    statStatus           := STATUS_SUBSEQUENT_CALL;
    statErrorAutoCleared := FALSE;
ELSE
    ;
END_IF;

statTorqueLimitingErrorOld := instTorqueLimiting.Error;
{END_REGION}

//----------------------------------------------------------------------------------------------
// Selection of StopOnError / implementation of fastStop
//----------------------------------------------------------------------------------------------
{REGION "STOP_ON_ERROR"}
// Check for stopping if error occurred during execution of motion commands
IF (statFBState = AXIS_STOP_ON_ERROR_SELECTION)
    THEN
    statBasicMotionState   := NO_SELECTION;
    statSupImpMotionState  := NO_SELECTION;
    statPassiveHomingState := NO_HOMING_ACTIVE;

    IF (configuration.generalSettings.stopOnError = TRUE)
        THEN
        // Read Statusword only when not already read out
        IF (tempStatusWord = 16#0)
            THEN
            tempStatusWord := axis.NcToPlc.StateDWord;
        END_IF;

        // Evaluate error
        IF tempStatusWord.0 THEN
            ; // Axis enabled
            IF (tempStatusWord.1 = TRUE) THEN
                ; // TO Alarm present
                statFBState := AXIS_MOTION;
            ELSE
                // No TO alarm present, set fastStop
                statBasicMotionState      := FAST_STOP_SELECTED;
                statFirstCycleBasicMotion := TRUE;
                statFBState               := AXIS_STOP_ON_ERROR_EXECUTION;
            END_IF;

        ELSE
            ; // Axis disabled
            statFBState := AXIS_MOTION;
        END_IF;

    ELSE
        // Dont StopOnError
        statFBState := AXIS_MOTION;
    END_IF;
END_IF;

// Implementation of fastStop
IF (statBasicMotionState = FAST_STOP_SELECTED) THEN
    // Additional feature: Load emergency stop dynamics (TO) if no valid dynamics are configured for fastStop
    {REGION "FASTSTOP SELECTED"}
    // Firstcycle of command
    IF (statFirstCycleBasicMotion = TRUE) THEN
        // Reset HALT command
        instHalt(Axis := axis,
                 Execute := FALSE);

        statFirstCycleDone := TRUE;
        // Check dynamics for fastStop
        // Load TO emergency Stop dynamics if value <=0 for deceleration is configured
        IF (configuration.fastStop.deceleration <= 0) // V1.0.2 Read TO emergencyStop deceleration only if fastStop.deceleration <= 0
            THEN
            // Invalid fastStop dynamics configured - read emergency stop dynamics from TO
            (*statDeceleration :=  axis.DynamicDefaults.EmergencyDeceleration;*)
            statDeceleration := configuration.fastStop.deceleration;
        ELSE
            // Valid fastStop dynamics configured
            statDeceleration := configuration.fastStop.deceleration;
        END_IF;

        statJerk              := configuration.fastStop.jerk;              // V1.0.2 Use always configuration for jerk value
        statAbortAcceleration := configuration.fastStop.abortAcceleration; // V1.0.2 Use always configuration
    END_IF;

    // Call of MC_Command
    instHalt(Axis := axis,
             Execute := (statBasicCommand.0 OR statFirstCycleBasicMotion),
             Deceleration := statDeceleration,
             (*AbortAcceleration :=  statAbortAcceleration,*)
             Jerk := statJerk);

    // Evaluate MC_Command
    IF (instHalt.Busy = FALSE) AND
        (instHalt.Error = FALSE) AND
        (instHalt.Done = FALSE) AND
        (instHalt.CommandAborted = FALSE)
        THEN
        // Return to NO_SELECTION if command finished
        statFBState          := AXIS_MOTION;
        statBasicMotionState := NO_SELECTION;

    ELSIF (instHalt.Done = TRUE)
        THEN
        IF (statFirstCycleDone = TRUE)
            THEN
            // Command is reset
            IF (instTorqueLimiting.Error = FALSE) // V1.00.03 Dont reset error is pending
                THEN
                // Reset status not if torquelimiting error is pending
                statStatus           := STATUS_SUBSEQUENT_CALL;
                statErrorAutoCleared := FALSE;
            END_IF;

            statFirstCycleDone := FALSE;
        END_IF;

    ELSIF (instHalt.Error = TRUE)
        THEN
        // Errorhandling
        statStatus                          := ERR_MC_HALT;
        statErrorAutoCleared                := TRUE;
        diagnostics                         := statDiagnostics;
        diagnostics.basicMotionState        := statBasicMotionState;
        diagnostics.superimposedMotionState := statSupImpMotionState;
        diagnostics.subfunctionStatus       := instHalt.ErrorId;

    ELSE
        ; // Command selected
    END_IF;

    // Write MC_Command outputs to internal variable
    statExeOfBasicMotion   := 0;
    statExeOfBasicMotion.0 := instHalt.Busy;
    statExeOfBasicMotion.1 := instHalt.Done;
    statExeOfBasicMotion.2 := instHalt.CommandAborted;
    statExeOfBasicMotion.3 := instHalt.Error;
    {END_REGION}
END_IF;

{END_REGION}
//----------------------------------------------------------------------------------------------
// Store values and reset variables
//----------------------------------------------------------------------------------------------
{REGION "STORE_AND_RESET"}
// Reset variables to determine first cycle of a new command
IF (statFirstCycleReset = TRUE) THEN
    statFirstCycleReset := FALSE;
END_IF;

IF (statFirstCycleHoming = TRUE) THEN
    statFirstCycleHoming := FALSE;
END_IF;

statHomingOld := tempHoming;

IF (statFirstCycleBasicMotion = TRUE) THEN
    statFirstCycleBasicMotion := FALSE;
END_IF;

statBasicCommandOld := statBasicCommand;

IF (statFirstCycleSupImpMotion = TRUE) THEN
    statFirstCycleSupImpMotion := FALSE;
END_IF;

statSupImpCommandOld := statSupImpCommand;

// Store last values for edge detection
statEnableOld          := enable;
statEnableAxisOld      := enableAxis;
statExtendedCommandOld := statExtendedCommand;
statPowerErrorOld      := instPower.Error;
{END_REGION}

//----------------------------------------------------------------------------------------------
// Writing outputs
//----------------------------------------------------------------------------------------------
{REGION "WRITING_OF_OUTPUTS"}
// Writing status outputs
resetActive := (statResetState = CMD_BUSY);

IF (statErrorUserCleared = TRUE) THEN
    ; // Reset variables at ErrorUserCleared
    statBasicMotionState       := NO_SELECTION;
    statExeOfBasicMotion       := NO_SELECTION;
    statSupImpMotionState      := NO_SELECTION;
    statExeOfSupImpMotionState := NO_SELECTION;
    statExeOfHoming            := NO_SELECTION;
END_IF;

IF (instPower.Status = TRUE)
    THEN
    // Axis enabled
    axisEnabled := TRUE;

ELSIF (instPower.Error = TRUE) AND (instPower.Status = FALSE)
    THEN
    // Reset status if error occurred
    axisEnabled := FALSE;

ELSIF (instPower.Busy = FALSE)
    THEN
    // Reset if MC_Power is not busy
    axisEnabled := FALSE;
ELSE
    ;
END_IF;

{REGION "WRITING_BASICMOTION_OUTPUTS"}
// Writing Busy, Done and Aborted outputs for basic motion commands
IF (statBasicMotionState > NO_SELECTION) AND (statBasicMotionState < ACTIVE_HOMING_SELECTED)
    THEN
    commandBusy    := statExeOfBasicMotion.0;
    commandDone    := statExeOfBasicMotion.1;
    commandAborted := statExeOfBasicMotion.2;
    inVelocity     := statExeOfBasicMotion.4;
    inSync         := statExeOfBasicMotion.7;
    startSync      := statExeOfBasicMotion.6;
ELSE
    commandBusy    := FALSE;
    commandDone    := FALSE;
    commandAborted := FALSE;
    inVelocity     := FALSE;
    inSync         := FALSE;
    startSync      := FALSE;
END_IF;

// Writing outputs up to LAxisCtrl_SpeedAxis
IF (statTorqueLimitingState = TORQUE_LIMTING_SELECTED)
// OR ( statTorqueLimitingState =  AUTOMATIC_MODE_CHANGE) V1.0.3 TorqueLimtinig = TRUE, only when respective value used 
    THEN
    torqueLimitingSelected := TRUE;
ELSE
    torqueLimitingSelected := FALSE;
END_IF;

inLimitation         := instTorqueLimiting.InLimitation;
fastStopSelected     := statBasicMotionState.0;
stopSelected         := statBasicMotionState.1;
jogSelected          := statBasicMotionState.2 OR statBasicMotionState.3;
moveVelocitySelected := statBasicMotionState.4;
// Writing outputs up to LAxisCtrl_PosAxis
inClamping          := instTorqueLimiting.InClamping;
posRelativeSelected := statBasicMotionState.5;
posAbsoluteSelected := statBasicMotionState.6;
// Writing outputs up to LAxisCtrl_SyncAxisRelGearing
gearInRelativeSelected := statBasicMotionState.7;
// Writing outputs up to LAxisCtrl_SyncAxisCamming
gearInAbsoluteSelected := statBasicMotionState.8;
camInSelected          := statBasicMotionState.9;
//inSimulation           := instSyncMotionSimulation.InSimulation;
{END_REGION}
{REGION "WRITING_HOMING_OUTPUTS"}
// Writing Busy, Done and Aborted outputs for homing
IF (statPassiveHomingState = STANDARD_HOMING)
    THEN
    homingSelected       := TRUE;
    homingCommandBusy    := statExeOfHoming.0;
    homingCommandDone    := statExeOfHoming.1;
    homingCommandAborted := statExeOfHoming.2;
ELSE
    IF (statBasicMotionState = ACTIVE_HOMING_SELECTED)
        THEN
        homingSelected       := TRUE;
        homingCommandBusy    := statExeOfBasicMotion.0;
        homingCommandDone    := statExeOfBasicMotion.1;
        homingCommandAborted := statExeOfBasicMotion.2;
    ELSE
        homingSelected       := FALSE;
        homingCommandBusy    := FALSE;
        homingCommandDone    := FALSE;
        homingCommandAborted := FALSE;
    END_IF;
END_IF;

{END_REGION}
{REGION "WRITING_SUPERIMPOSED_OUTPUTS"}
// Writing outputs for superimposed motion commands
IF (statSupImpMotionState <> NO_SELECTION)
    THEN
    superimposedBusy    := statExeOfSupImpMotionState.0;
    superimposedDone    := statExeOfSupImpMotionState.1;
    superimposedAborted := statExeOfSupImpMotionState.2;
ELSE
    superimposedBusy    := FALSE;
    superimposedDone    := FALSE;
    superimposedAborted := FALSE;
END_IF;

posSuperimposedSelected := statSupImpMotionState.0;
phasingSelected         := statSupImpMotionState.1;
{END_REGION}
{END_REGION}

//----------------------------------------------------------------------------------------------
// Error handling 
//----------------------------------------------------------------------------------------------
{REGION "ERROR_HANDLING"}
IF statErrorUserCleared THEN
    valid              := FALSE;
    busy               := TRUE;
    error              := TRUE;
    status             := statStatus;
    diagnostics.status := statStatus;

ELSIF statErrorAutoCleared THEN
    valid              := FALSE;
    busy               := TRUE;
    error              := TRUE;
    status             := statStatus;
    diagnostics.status := statStatus;

ELSE
    // Process normal output values
    valid  := TRUE;
    error  := FALSE;
    status := statStatus;
END_IF;

{END_REGION}

END_FUNCTION_BLOCK

(* stored: Version 1.1.0.1
   POU FB_ComplexAxisControl: Id {d5fd03af-b1eb-4c28-9290-c4b09e920204}, SpecialFunc None *)
